Staubli VAL3: Numerisation.dtx

bool bAcquisitionStarted = true
bool bOverrun
jointRx jCurrentJoint = {j1=-9.566067, j2=37.23348, j3=99.811939, j4=1.059303e-14, j5=42.95458, j6=-9.566067}
jointRx jCurrentJointError = {j1=0.00111051, j2=-0.000418031, j3=-0.000552065, j4=-0.00000679927, j5=-0.000103346, j6=0.000911689}
jointRx jInitialPosition = {j2=37.32, j3=99.65, j5=43.03}
jointRx jInitialPositionRepos = {j2=28.35, j3=97.17, j5=54.5}
jointRx jRobotZeroPosition = {j6=90}
mdesc mNomSpeed
num nBinaryPositionArray[24]
  [0] = 68
  [1] = 21
  [2] = 43
  [3] = 8
  [4] = 194
  [5] = 71
  [6] = 116
  [7] = 129
  [8] = 194
  [9] = 145
  [10] = 94
  [11] = 130
  [12] = 57
  [13] = 16
  [14] = 130
  [15] = 243
  [16] = 195
  [17] = 51
  [18] = 255
  [19] = 204
  [20] = 57
  [21] = 54
  [22] = 234
  [23] = 129
num nBinaryPositionArrayIndex
num nCurrentPositionArray[6]
  [0] = 596.672343
  [1] = -49.863772
  [2] = -72.684587
  [3] = 0.000137817
  [4] = -179.999203
  [5] = 0.000174442
num nMaxHorizontal = 1000
num nMaxRotation = 180
num nMaxVertical = 950
num nMinHorizontal = -1000
num nMinRotation = -180
num nMinVertical = -883.44
num nNextPositionX = 737.67
num nReceivedByte = 10
num nScanningLength = 200
num nScanningLineNumber = 5
num nScanningWidth = 200
pointRx pCircle = {x=497.67, y=50, z=-72.68, rx=-180, rz=-180, shoulder=sfree, elbow=efree, wrist=wfree, fatherId=world[0]}
pointRx pCurrentPosition = {x=596.760773, y=-49.877677, z=-72.686767, rx=0.000182979, ry=-179.998942, rz=0.000203803, shoulder=lefty, elbow=epositive, wrist=wpositive, fatherId=world[0]}
pointRx pInitialPosition = {x=597.67, y=50, z=-72.68, rx=-180, rz=-180, shoulder=sfree, elbow=efree, wrist=wfree, fatherId=world[0]}
pointRx pInitialPositionRepos = {x=597.67, y=50, z=27.32, rx=-180, rz=-180, shoulder=sfree, elbow=efree, wrist=wfree, fatherId=world[0]}
pointRx pNextPosition = {x=597.67, y=-50, z=-72.68, rx=-180, rz=-180, shoulder=sfree, elbow=efree, wrist=wfree, fatherId=world[0]}
pointRx pRobotZeroPosition = {x=50, y=50, z=950, shoulder=sfree, elbow=efree, wrist=wfree, fatherId=world[0]}
public sio sioSockets_c1 = {link=UdpSocket\c1}
